SUBAPPLICATION Uebung_071_AX (* WBSD auf UT ausgeben, Q1 Schalten wenn Speed > 0 (Adapter Version) *)
  (* Standard: 61499-2; Description: Copyright (c) 2023-2026 Meisterschulen am Ostbahnhof This program and the accompanying materials are made available under the terms of the Eclipse Public License 2.0 which is available at https://www.eclipse.org/legal/epl-2.0/ SPDX-License-Identifier: EPL-2.0 *)
  (* Version 1.0, 2026-04-19, Franz Höpfinger, Meisterschulen am Ostbahnhof, initial API and implementation (Adapter Version of Uebung_071) *)
  PACKAGE Uebungen;
  IMPORT Uebungen::const::UT::TECU::DefaultPool_TECU::NumberVariable_Wheel_based_machine_speed;
  IMPORT logiBUS::io::DQ::logiBUS_DO::Output_Q1;
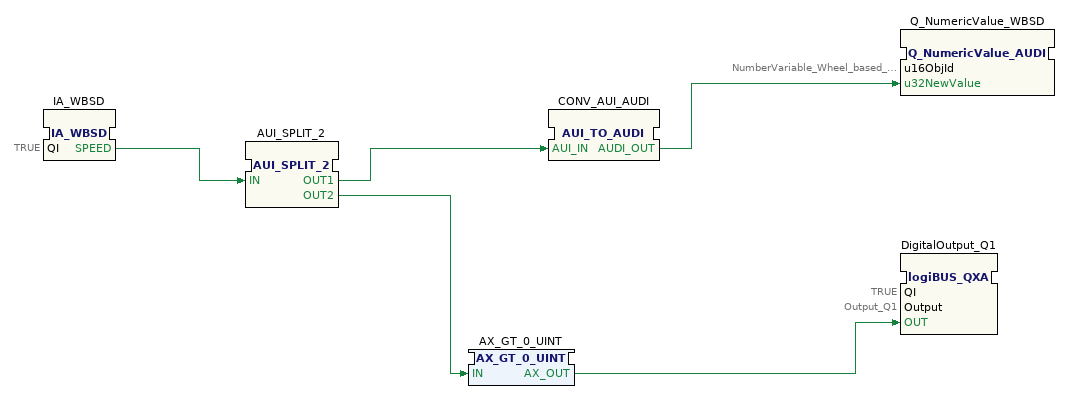
  FBS
    IA_WBSD : isobus::tecu::IA_WBSD(QI := TRUE);
    Q_NumericValue_WBSD : isobus::UT::Q::Q_NumericValue_AUDI(u16ObjId := NumberVariable_Wheel_based_machine_speed);
    DigitalOutput_Q1 : logiBUS::io::DQ::logiBUS_QXA(QI := TRUE, Output := Output_Q1);
    CONV_AUI_AUDI : adapter::conversion::unidirectional::AUI_TO_AUDI;
    AUI_SPLIT_2 : adapter::events::unidirectional::AUI_SPLIT_2;
  END_FBS
  SUBAPPS
    AX_GT_0_UINT : MyLib::sys::AX_GT_0_UINT;
  END_SUBAPPS
  ADAPTER_CONNECTIONS
    AUI_SPLIT_2.OUT1 TO CONV_AUI_AUDI.AUI_IN;
    CONV_AUI_AUDI.AUDI_OUT TO Q_NumericValue_WBSD.u32NewValue;
    IA_WBSD.SPEED TO AUI_SPLIT_2.IN;
    AUI_SPLIT_2.OUT2 TO AX_GT_0_UINT.IN;
    AX_GT_0_UINT.AX_OUT TO DigitalOutput_Q1.OUT;
  END_CONNECTIONS
END_SUBAPPLICATION
